(* Logix 5000 project; controller DIMTER vendor 1 type 14 code 77 rev 15.4; software revision 15.01 *)
// Dimter PLC Upgrade

TASK MainTask (continuous, watchdog 500 ms) : MainProgram

MODULES
   Controller : vendor 1 type 14 code 77 (CompactLogixL32EController 0, rev 15.4)
      LocalENB : 1769-L32E Ethernet Port (CompactLogixL32Ethernet 1, Ethernet 10.1.1.1, rev 15.1)
      Local : CompactBus (CompactVirtualAdapter 3, rev 15.1, Input RPI 2 ms)
          : 1769-IQ32 (Compact 1, rev 3.1, Input RPI 2 ms)
          : 1769-IQ32 (Compact 2, rev 3.1, Input RPI 2 ms)
          : 1769-IQ32 (Compact 3, rev 3.1, Input RPI 2 ms)
          : 1769-OW16 (Compact 4, rev 1.1, Output RPI 2 ms)
          : 1769-OW16 (Compact 5, rev 1.1, Output RPI 2 ms)
          : 1769-OW16 (Compact 6, rev 1.1, Output RPI 2 ms)
          : 1769-OW16 (Compact 7, rev 1.1, Output RPI 2 ms)
END_MODULES

TYPE FaultRecord :
STRUCT
   TimeLow : DINT;
   TimeHigh : DINT;
   Type : INT;
   Code : INT;
   Info : DINT[8];
END_STRUCT
END_TYPE

TYPE RTC :   // Real Time Clock
STRUCT
   Year : DINT;   // RTC Year
   Month : DINT;   // RTC Month
   Day : DINT;   // RTC Day
   Hour : DINT;   // RTC Hour
   Minute : DINT;   // RTC Minute
   Second : DINT;   // RTC Second
   uSecond : DINT;   // RTC uSecond
   DayOfWeek : DINT;   // RTC Day Of Week
END_STRUCT
END_TYPE

VAR_GLOBAL   (* controller tags *)
   A120 : ALIAS FOR Local:4:O.Data.0;   // O:4.0/0 A12.0 Buffer Selection1
   A121 : ALIAS FOR Local:4:O.Data.1;   // O:4.0/1 A12/1 Buffer Selection 2
   A122 : ALIAS FOR Local:4:O.Data.2;   // O:4.0/2 A12.2 Reset Failure
   A123 : ALIAS FOR Local:4:O.Data.3;   // O:4.0/3 A12.3 Reset Buffer
   A124 : ALIAS FOR Local:4:O.Data.4;   // O:4.0/4 A12.4 Spare
   A125 : ALIAS FOR Local:4:O.Data.5;   // O:4.0/5 A12.5 Spare
   A126 : ALIAS FOR Local:4:O.Data.6;   // O:4.0/6 A12.6 Spare
   A127 : ALIAS FOR Local:4:O.Data.7;   // O:4.0/7 A12.7 Spare
   A130 : ALIAS FOR Local:4:O.Data.8;   // O:4.0/8 A13.0 Failure Conveyor
   A131 : ALIAS FOR Local:4:O.Data.9;   // O:4.0/9 A13.1 Failure Saw 1
   A132 : ALIAS FOR Local:4:O.Data.10;   // O:4.0/10 A13.2 Failure Saw 2
   A133 : ALIAS FOR Local:4:O.Data.11;   // O:4.0/11 A13.3 Defect Measuring Computer
   A134 : ALIAS FOR Local:4:O.Data.12;   // O:4.0/12 A13.4 Safety Barrier Transfer Station
   A135 : ALIAS FOR Local:4:O.Data.13;   // O:4.0/13 A13.5 Unknown
   A136 : ALIAS FOR Local:4:O.Data.14;   // O:4.0/14 A136 Unknown
   A137 : ALIAS FOR Local:4:O.Data.15;   // O:4.0/15 A137 Safety Barrier Transfer Station
   A140 : ALIAS FOR Local:5:O.Data.0;   // O:5.0/0 A140 Chain Ejector Fast Left
   A141 : ALIAS FOR Local:5:O.Data.1;   // O:5.0/1 A141 Chain Ejector Slow Left
   A142 : ALIAS FOR Local:5:O.Data.2;   // O:5.0/2 A142 Raise Rake 1
   A143 : ALIAS FOR Local:5:O.Data.3;   // O:5.0/3 A143 Brake Cross Conveyor Front of Saw 1
   A144 : ALIAS FOR Local:5:O.Data.4;   // O:5.0/4 A144 Cross Feed 1 Fast Fwd
   A145 : ALIAS FOR Local:5:O.Data.5;   // O:5.0/5 A145 Cross Feed 1 Slow Fwd
   A146 : ALIAS FOR Local:5:O.Data.6;   // O:5.0/6 A146 Cross Feed 1 Fast Rev
   A147 : ALIAS FOR Local:5:O.Data.7;   // O:5.0/7 A147 Infeed Roller Saw 1
   A150 : ALIAS FOR Local:5:O.Data.8;   // O:5.0/8 A15.0 Rollcase 1 VSD Run Enable
   A151 : ALIAS FOR Local:5:O.Data.9;   // O:5.0/9 A15.1 Jog Rollcase 1 Set Speed
   A152 : ALIAS FOR Local:5:O.Data.10;   // O:5.0/10 A15.2 Forward Rotation Rollcase 1
   A153 : ALIAS FOR Local:5:O.Data.11;   // O:5.0/11 A15.3 Brake Rollcase Front of Saw 1
   A154 : ALIAS FOR Local:5:O.Data.12;   // O:5.0/12 A15.4 Rollcase 2 VSD Run Enable
   A155 : ALIAS FOR Local:5:O.Data.13;   // O:5.0/13 A155 Jog Rollcase 2 Set Speed
   A156 : ALIAS FOR Local:5:O.Data.14;   // O:5.0/14 A156 Forward Rotation Rollcase 2
   A157 : ALIAS FOR Local:5:O.Data.15;   // O:5.0/15 A157 Brake Rollcase 2
   A160 : ALIAS FOR Local:6:O.Data.0;   // O:6.0/0 A16.0 Chain Ejector Fast Right
   A161 : ALIAS FOR Local:6:O.Data.1;   // O:6.0/1 A16.1 Chain Ejector Slow Right
   A162 : ALIAS FOR Local:6:O.Data.2;   // O:6.0/2 A16.2 Rake 2
   A163 : ALIAS FOR Local:6:O.Data.3;   // O:6.0/3 A16.3 Brake Cross Conveyor Front of Saw 2
   A164 : ALIAS FOR Local:6:O.Data.4;   // O:6.0/4 A16.4 Cross Feed 2 Fast Fwd
   A165 : ALIAS FOR Local:6:O.Data.5;   // O:6.0/5 A16.5 Cross Feed 2 Slow Fwd
   A166 : ALIAS FOR Local:6:O.Data.6;   // O:6.0/6 A16.6 Cross Feed 2 Fast Rev
   A167 : ALIAS FOR Local:6:O.Data.7;   // O:6.0/7 A16.7 Infeed Roller Saw 2
   A170 : ALIAS FOR Local:6:O.Data.8;   // O:6.0/8 A17.0 Infeed Measuring Slot Weinig Release Workpiece to Demand
   A171 : ALIAS FOR Local:6:O.Data.9;   // O:6.0/9 A17.1 Conveyor Measuring Slot Weinig Feed to Switch On
   A172 : ALIAS FOR Local:6:O.Data.10;   // O:6.0/10 A17.2 Chain Ejector Brake
   A173 : ALIAS FOR Local:6:O.Data.11;   // O:6.0/11 A17.3 Spare
   A174 : ALIAS FOR Local:6:O.Data.12;   // O:6.0/12 A17.4 Spare
   A175 : ALIAS FOR Local:6:O.Data.13;   // O:6.0/13 A17.5 Spare
   A176 : ALIAS FOR Local:6:O.Data.14;   // O:6.0/14 A17.6 Spare
   A177 : ALIAS FOR Local:6:O.Data.15;   // O:6.0/15 A17.7 Spare
   A180 : ALIAS FOR Local:7:O.Data.0;   // O:7.0/0 A18.0 VSD Feed Contactor Rollcase 1
   A181 : ALIAS FOR Local:7:O.Data.1;   // O:7.0/1 A18.1 VSD Feed Contactor Rollcase 2
   A182 : ALIAS FOR Local:7:O.Data.2;   // O:7.0/2 A18.2 Infeed Roller Measuring Station
   A183 : ALIAS FOR Local:7:O.Data.3;   // O:7.0/3 A18.3 Unknown
   A184 : ALIAS FOR Local:7:O.Data.4;   // O:7.0/4 A18.4 Waste Belt Conveyor 1
   A185 : ALIAS FOR Local:7:O.Data.5;   // O:7.0/5 A18.5 Waste Belt Conveyor 2
   A186 : ALIAS FOR Local:7:O.Data.6;   // O:7.0/6 A18.6 Cross Belt 1
   A187 : ALIAS FOR Local:7:O.Data.7;   // O:7.0/7 A18.7 Cross Belt 2
   A190 : ALIAS FOR Local:7:O.Data.8;   // O:7.0/8 A19.0 Spare
   A191 : ALIAS FOR Local:7:O.Data.9;   // O:7.0/9 A19.1 Spare
   A192 : ALIAS FOR Local:7:O.Data.10;   // O:7.0/10 A19.2 Spare
   A193 : ALIAS FOR Local:7:O.Data.11;   // O:7.0/11 A19.3 Spare
   A194 : ALIAS FOR Local:7:O.Data.12;   // O:7.0/12 A19.4 Spare
   A195 : ALIAS FOR Local:7:O.Data.13;   // O:7.0/13 A19.5 Spare
   A196 : ALIAS FOR Local:7:O.Data.14;   // O:7.0/14 A19.6 Spare
   A197 : ALIAS FOR Local:7:O.Data.15;   // O:7.0/15 A19.7 Spare
   BitArrayFromHMI : INT[100]; {produced}
   BitArrayToHMI : INT[130] := ([6] := 14, [7] := 15);
   BitsFromHMI : BOOL[128];   // Bits From HMI
   Debounce : TIMER[30] := ([0].PRE := 100, [1].PRE := 100);   // Debounce Timers
        [0]   // PE Infeed Saw 1 Debounce
        [1]   // PE Roller 1 Debounce
   Delay : TIMER[30] := ([0].PRE := 300, [1].PRE := 300, [2].PRE := 100);   // Delay Timers
        [0]   // Saw 1 Cutting Delay
        [1]   // Saw 2 Cutting Delay
   E00 : ALIAS FOR Local:1:I.Data.0;   // I:1.0/0 E0.0 Control Power On
   E01 : ALIAS FOR Local:1:I.Data.1;   // I:1.0/1 E0.1 Saw Hood 1 Closed
   E02 : ALIAS FOR Local:1:I.Data.2;   // I:1.0/2 E0.2 Saw Motor 1 On
   E03 : ALIAS FOR Local:1:I.Data.3;   // I:1.0/3 E0.3 Release - Feed Saw 1
   E04 : ALIAS FOR Local:1:I.Data.4;   // I:1.0/4 E0.4 Failure Saw 1
   E05 : ALIAS FOR Local:1:I.Data.5;   // I:1.0/5 E0.5 Failure Chain Ejector
   E06 : ALIAS FOR Local:1:I.Data.6;   // I:1.0/6 E0.6 Failure Conveyor in Front of Saw 1
   E07 : ALIAS FOR Local:1:I.Data.7;   // I:1.0/7 E0.7 Failure Conveyor in Front of Saw 2
   E10 : ALIAS FOR Local:1:I.Data.8;   // I:1.0/8 E1.0 Failure Weinig Conveyor
   E100 : ALIAS FOR Local:3:I.Data.16;   // I:3.1/0 E10.0 Sorting Ejector Sorting 1
   E101 : ALIAS FOR Local:3:I.Data.17;   // I:3.1/1 E10.1 Sorting Ejector 2 Sorting 1
   E102 : ALIAS FOR Local:3:I.Data.18;   // I:3.1/2 E10.2 Sorting Ejector 3 Sorting 1
   E103 : ALIAS FOR Local:3:I.Data.19;   // I:3.1/3 E10.3 Sorting Ejector 1 Sorting 2
   E104 : ALIAS FOR Local:3:I.Data.20;   // I:3.1/4 E10.4 Sorting Ejector 2 Sorting 2
   E105 : ALIAS FOR Local:3:I.Data.21;   // I:3.1/5 E10.5 Sorting Ejector 3 Sorting 2
   E106 : ALIAS FOR Local:3:I.Data.22;   // I:3.1/6 E10.6 Cross Belt 1 Cyclewise Continuous Running
   E107 : ALIAS FOR Local:3:I.Data.23;   // I:3.1/7 E10.7 ???
   E11 : ALIAS FOR Local:1:I.Data.9;   // I:1.0/9 E1.1 Saw Hood 2 Closed
   E110 : ALIAS FOR Local:3:I.Data.24;   // I:3.1/8 E11.0 Cross Belt 1 Footswitch (Removed)
   E111 : ALIAS FOR Local:3:I.Data.25;   // I:3.1/9 E11.1 Cross Belt 2 Cyclewise Continuous Running
   E112 : ALIAS FOR Local:3:I.Data.26;   // I:3.1/10 E11.2 ???
   E113 : ALIAS FOR Local:3:I.Data.27;   // I:3.1/11 E11.3 Cross Belt 2 Footswitch (Removed)
   E114 : ALIAS FOR Local:3:I.Data.28;   // I:3.1/12 E11.4 Transfer Station On
   E115 : ALIAS FOR Local:3:I.Data.29;   // I:3.1/13 E11.5 Cross Feed Manual Fwd-Rev
   E116 : ALIAS FOR Local:3:I.Data.30;   // I:3.1/14 E11.6 ???
   E117 : ALIAS FOR Local:3:I.Data.31;   // I:3.1/1 5 E11.7 Acknowledge Failure
   E12 : ALIAS FOR Local:1:I.Data.10;   // I:1.0/10 E1.2 Saw Motor 2 On
   E13 : ALIAS FOR Local:1:I.Data.11;   // I:1.0/11 E1.3 Release - Feed Saw 2
   E14 : ALIAS FOR Local:1:I.Data.12;   // I:1.0/12 E1.4 Failure Saw 2
   E15 : ALIAS FOR Local:1:I.Data.13;   // I:1.0/13 E1.5 Data Ready At Saw
   E16 : ALIAS FOR Local:1:I.Data.14;   // I:1.0/14 E1.6 Release Optimisation
   E17 : ALIAS FOR Local:1:I.Data.15;   // I:1.0/15 E1.7 Defect Measuring Computer
   E20 : ALIAS FOR Local:1:I.Data.16;   // I:1.1/0 E2.0 Protection Hood Measuring System
   E21 : ALIAS FOR Local:1:I.Data.17;   // I:1.1/1 E2.1 Spare
   E22 : ALIAS FOR Local:1:I.Data.18;   // I:1.1/2 E2.2 Frequency Converter Rollcase in Front of Saw 1 Ready For Operation
   E23 : ALIAS FOR Local:1:I.Data.19;   // I:1.1/3 E2.3 Frequency Converter Rollcase in Front of Saw 2 Ready For Operation
   E24 : ALIAS FOR Local:1:I.Data.20;   // I:1.1/4 E2.4 Emergency Shutdown Internal
   E25 : ALIAS FOR Local:1:I.Data.21;   // I:1.1/5 E2.5 Emergency Shutdown External
   E26 : ALIAS FOR Local:1:I.Data.22;   // I:1.1/6 E2.6 Safety Barrier at Transfer Station Closed
   E27 : ALIAS FOR Local:1:I.Data.23;   // I:1.1/7 E2.7 Reset Safety Barrier at Transfer Station
   E30 : ALIAS FOR Local:1:I.Data.24;   // I:1.1/8 E3.0 Spare
   E31 : ALIAS FOR Local:1:I.Data.25;   // I:1.1/9 E3.1 PE in Front of Measuring Station
   E32 : ALIAS FOR Local:1:I.Data.26;   // I:1.1/10 E3.2 Start Measurement Measurement Station
   E33 : ALIAS FOR Local:1:I.Data.27;   // I:1/1/11 E3.3 PE Behind Measurement Station
   E34 : ALIAS FOR Local:1:I.Data.28;   // I:1.1/12 E3.4 Spare
   E35 : ALIAS FOR Local:1:I.Data.29;   // I:1.1/13 E3.5 Spare
   E36 : ALIAS FOR Local:1:I.Data.30;   // I:1.1/14 E3.6 Spare
   E37 : ALIAS FOR Local:1:I.Data.31;   // I:1.1/15 E3.7 Spare
   E40 : ALIAS FOR Local:2:I.Data.0;   // I:2.0/0 E4.0 Chain Ejector Manual Left
   E41 : ALIAS FOR Local:2:I.Data.1;   // I:2.0/1 E4.1 Cross Feed 1 Manual Fwd - Rev
   E42 : ALIAS FOR Local:2:I.Data.2;   // I:2.0/2 E4.2 Cross Feed 1 Manual Fwd - Rev
   E43 : ALIAS FOR Local:2:I.Data.3;   // I:2.0/3 E4.3 Infeed Saw 1 On
   E44 : ALIAS FOR Local:2:I.Data.4;   // I:2.0/4 E4.4 Waste Conveyor Belt On
   E45 : ALIAS FOR Local:2:I.Data.5;   // I:2.0/5 E4.5 Transfer Station in Front of Saw On
   E46 : ALIAS FOR Local:2:I.Data.6;   // I:2.0/6 E4.6 Acknowledge Failure
   E47 : ALIAS FOR Local:2:I.Data.7;   // I:2.0/7 E4.7 Lamp Test
   E50 : ALIAS FOR Local:2:I.Data.8;   // I:2.0/8 E5.0 Chain Ejector Manual Right
   E51 : ALIAS FOR Local:2:I.Data.9;   // I:2.0/9 E5.1 Cross Feed 2 Manual Fwd - Rev
   E52 : ALIAS FOR Local:2:I.Data.10;   // I:2.0/10 E5.2 Cross Feed 2 Manual Fwd - Rev
   E53 : ALIAS FOR Local:2:I.Data.11;   // I:2.0/11 E5.3 Infeed Saw 2 On
   E54 : ALIAS FOR Local:2:I.Data.12;   // I:2.0/12 E5.4 Measuring Station On
   E55 : ALIAS FOR Local:2:I.Data.13;   // I:2.0/13 E5.5 Reset Defect Measuring Computer
   E56 : ALIAS FOR Local:2:I.Data.14;   // I:2.0/14 E5.6 Reset Buffer Measuring Computer
   E57 : ALIAS FOR Local:2:I.Data.15;   // I:2.0/15 E5.7 Conveyor Measuring Station Manual
   E60 : ALIAS FOR Local:2:I.Data.16;   // I:2.1/0 E6.0 Spare
   E61 : ALIAS FOR Local:2:I.Data.17;   // I:2.1/1 E6.1 PE Infeed Saw 1
   E62 : ALIAS FOR Local:2:I.Data.18;   // I:2.1/2 E6.2 PE Front of Saw 1
   E63 : ALIAS FOR Local:2:I.Data.19;   // I:2.1/3 E6.3 PE Roller 1
   E64 : ALIAS FOR Local:2:I.Data.20;   // I:2.1/4 E6.4 Feed Saw 1 On
   E65 : ALIAS FOR Local:2:I.Data.21;   // I:2.1/5 E6.5 Spare
   E66 : ALIAS FOR Local:2:I.Data.22;   // I:2.1/6 E6.6 Release Chain Ejector Saw 1 Cross Feed
   E67 : ALIAS FOR Local:2:I.Data.23;   // I:2.1/7 E6.7 PE Cross Feed 1 Waiting Position
   E70 : ALIAS FOR Local:2:I.Data.24;   // I:2.1/8 E7.0 PE Chain Ejector Home Position Left
   E71 : ALIAS FOR Local:2:I.Data.25;   // I:2.1/9 E7.1 PE Chain Ejector Initial Position Left Front
   E72 : ALIAS FOR Local:2:I.Data.26;   // I:2.1/10 E7.2 Stop Rollcase 1
   E73 : ALIAS FOR Local:2:I.Data.27;   // I:2.1/11 E7.3 Cross Feed 1 Down
   E74 : ALIAS FOR Local:2:I.Data.28;   // I:2.1/12 E7.4 Cross Feed 1 Up
   E75 : ALIAS FOR Local:2:I.Data.29;   // I:2.1/13 E7.5 Cross Feed 1 Initial Position
   E76 : ALIAS FOR Local:2:I.Data.30;   // I:2.1/14 E7.6 PE Cross Feed 1 Slow Fwd
   E77 : ALIAS FOR Local:2:I.Data.31;   // I:2.1/15 E7.7 Cross Feed 1 at Front
   E80 : ALIAS FOR Local:3:I.Data.0;   // I:3.0/0 E8.0 Spare
   E81 : ALIAS FOR Local:3:I.Data.1;   // I:3.0/1 E8.1 PE Infeed Saw 2
   E82 : ALIAS FOR Local:3:I.Data.2;   // I:3.0/2 E8.2 PE Front of Saw 2
   E83 : ALIAS FOR Local:3:I.Data.3;   // I:3.0/3 E8.3 PE Roller 2
   E84 : ALIAS FOR Local:3:I.Data.4;   // I:3.0/4 E8.4 Feed Saw 2 On
   E85 : ALIAS FOR Local:3:I.Data.5;   // I:3.0/5 E8.5 Spare
   E86 : ALIAS FOR Local:3:I.Data.6;   // I:3.0/6 E8.6 Release (Enable) Chain Ejector Saw 2 Cross Feed
   E87 : ALIAS FOR Local:3:I.Data.7;   // I:3.0/7 E8.7 PE Cross Feed 2 Waiting Position
   E90 : ALIAS FOR Local:3:I.Data.8;   // I:3.0/8 E9.0 PE Chain Ejector Initial Position Right
   E91 : ALIAS FOR Local:3:I.Data.9;   // I:3.0/9 E9.1 PE Chain Ejector Initial Position Right Front
   E92 : ALIAS FOR Local:3:I.Data.10;   // I:3.0/10 E9.2 Stop Rollcase 2
   E93 : ALIAS FOR Local:3:I.Data.11;   // I:3.0/11 E9.3 Cross Feed 2 Down
   E94 : ALIAS FOR Local:3:I.Data.12;   // I:3.0/12 E9.4 Cross Feed 2 Up
   E95 : ALIAS FOR Local:3:I.Data.13;   // I:3.0/13 E9.5 Cross Feed 2 Home Position
   E96 : ALIAS FOR Local:3:I.Data.14;   // I:3.0/14 E9.6 PE Cross Feed 2 Slow Fwd
   E97 : ALIAS FOR Local:3:I.Data.15;   // I:3.0/15 E9.7 Cross Feed 2 at Front
   Faults : BOOL[224] := ([0] := 1, [14] := 1);   // Fault Array
   FirstPass : BOOL;   // On for First Scan
   HMI_Bits : BOOL[2016] := ([20] := 1, [44] := 1, [111] := 1, [112] := 1, [113] := 1, [114] := 1, [115] := 1, [118] := 1, [119] := 1, [120] := 1, [121] := 1, [122] := 1, [316] := 1, [330] := 1, [357] := 1, [1033] := 1); {produced}   // Bits to HMI
   HMI_IntWords : INT[200] := ([0] := 38, [2] := 323, [3] := 268, [4] := 591, [30] := 427, [31] := 576, [32] := 1003, [34] := 403, [35] := 649, [36] := 1052, [38] := 1543, [39] := 1599, [40] := 3142, [42] := 374, [43] := 450, [44] := 824, [46] := 1739, [47] := 1704, [48] := 3443, [54] := 2187, [55] := 2818, [56] := 5005, [58] := 427, [59] := 576, [60] := 1003, [62] := 403, [63] := 649, [64] := 1052, [66] := 1543, [67] := 1599, [68] := 3142, [70] := 374, [71] := 450, [72] := 824, [74] := 1739, [75] := 1704, [76] := 3443, [82] := 2187, [83] := 2818, [84] := 5005); {produced}   // Integer Words to HMI
        [0]   // Screen Command to HMI
        [1]   // Screen Displayed From HMI
        [2]   // Shift A Monday Saw 1 Total
        [3]   // Shift A Monday Saw 2 Total
        [4]   // Shift A Monday Grand Total
        [5]   // Shift A Monday Total Faults
        [6]   // Shift A Tuesday Saw 1 Total
        [7]   // Shift A Tuesday Saw 2 Total
        [8]   // Shift A Tuesday Grand Total
        [9]   // Shift A Tuesday Total Faults
        [10]   // Shift A Wednesday Saw 1 Total
        [11]   // Shift A Wednesday Saw 2 Total
        [12]   // Shift A Wednesday Grand Total
        [13]   // Shift A Wednesday Total Faults
        [14]   // Shift A Thursday Saw 1 Total
        [15]   // Shift A Thursday Saw 2 Total
        [16]   // Shift A Thursday Grand Total
        [17]   // Shift A Thursday Total Faults
        [18]   // Shift A Friday Saw 1 Total
        [19]   // Shift A Friday Saw 2 Total
        [20]   // Shift A Friday Grand Total
        [21]   // Shift A Friday Total Faults
        [22]   // Shift A Saturday Saw 1 Total
        [23]   // Shift A Saturday Saw 2 Total
        [24]   // Shift A Saturday Grand Total
        [25]   // Shift A Saturday Total Faults
        [26]   // Shift A Sunday Saw 1 Total
        [27]   // Shift A Sunday Saw 2 Total
        [28]   // Shift A Sunday Grand Total
        [29]   // Shift A Sunday Total Faults
        [30]   // Shift B Monday Saw 1 Total
        [31]   // Shift B Monday Saw 2 Total
        [32]   // Shift B Monday Grand Total
        [33]   // Shift B Monday Total Faults
        [34]   // Shift B Tuesday Saw 1 Total
        [35]   // Shift B Tuesday Saw 2 Total
        [36]   // Shift B Tuesday Grand Total
        [37]   // Shift B Tuesday Total Faults
        [38]   // Shift B Wednesday Saw 1 Total
        [46]   // Shift B Friday Saw 1 Total
        [47]   // Shift B Friday Saw 2 Total
        [43]   // Shift B Thursday Saw 2 Total
        [48]   // Shift B Friday Grand Total
        [39]   // Shift B Wednesday Saw 2 Total
        [40]   // Shift B Wednesday Grand Total
        [41]   // Shift B Wednesday Total Faults
        [42]   // Shift B Thursday Saw 1 Total
        [44]   // Shift B Thursday Grand Total
        [45]   // Shift B Thursday Total Faults
        [49]   // Shift B Friday Total Faults
        [50]   // Shift B Saturday Saw 1 Total
        [51]   // Shift B Saturday Saw 2 Total
        [52]   // Shift B Saturday Grand Total
        [53]   // Shift B Saturday Total Faults
        [54]   // Shift B Sunday Saw 1 Total
        [55]   // Shift B Sunday Saw 2 Total
        [56]   // Shift B Sunday Grand Total
        [57]   // Shift B Sunday Total Faults
        [58]   // Shift C Monday Saw 1 Total
        [59]   // Shift C Monday Saw 2 Total
        [60]   // Shift C Monday Grand Total
        [61]   // Shift C Monday Total Faults
        [62]   // Shift C Tuesday Saw 1 Total
        [63]   // Shift C Tuesday Saw 2 Total
        [64]   // Shift C Tuesday Grand Total
        [65]   // Shift C Tuesday Total Faults
        [66]   // Shift C Wednesday Saw 1 Total
        [67]   // Shift C Wednesday Saw 2 Total
        [68]   // Shift C Wednesday Grand Total
        [69]   // Shift C Wednesday Total Faults
        [70]   // Shift C Thursday Saw 1 Total
        [71]   // Shift C Thursday Saw 2 Total
        [72]   // Shift C Thursday Grand Total
        [73]   // Shift C Thursday Total Faults
        [74]   // Shift C Friday Saw 1 Total
        [75]   // Shift C Friday Saw 2 Total
        [76]   // Shift C Friday Grand Total
        [77]   // Shift C Friday Total Faults
        [78]   // Shift C Saturday Saw 1 Total
        [79]   // Shift C Saturday Saw 2 Total
        [80]   // Shift C Saturday Grand Total
        [81]   // Shift C Saturday Total Faults
        [82]   // Shift C Sunday Saw 1 Total
        [83]   // Shift C Sunday Saw 2 Total
        [84]   // Shift C Sunday Grand Total
        [85]   // Shift C Sunday Total Faults
   HMI_RealWords : REAL[20]; {produced}   // Real Words to HMI Transfer file
        [1]   // Saw 2 Hourmeter
        [4]   // Cross Feed 1 Hourmeter
        [7]   // Waste Belt 1 Hourmeter
        [2]   // Infeed Rolls 1 Hourmeter
        [0]   // Saw 1 Hourmeter
        [3]   // Infeed Rolls 2 Hourmeter
        [5]   // Cross Feed 2 Hourmeter
        [6]   // Chain Ejector Hourmeter
        [8]   // Waste Belt 2 Hourmeter
        [9]   // Cross Belt 1 Hourmeter
        [10]   // Cross Belt 2 Hourmeter
   HMI_TimerPresets : INT[100]; {produced}   // Timer Preset Data from HMI
   IntsFromHMI : INT[100] := ([0] := 5, [2] := 13, [4] := 5, [6] := 13, [8] := 5, [10] := 13, [12] := 5, [14] := 13, [16] := 5, [18] := 13, [28] := 13, [30] := 23, [32] := 13, [34] := 23, [36] := 13, [38] := 23, [40] := 13, [42] := 23, [44] := 13, [46] := 23, [56] := 21, [58] := 5, [60] := 21, [62] := 5, [63] := 21, [65] := 5, [66] := 21, [68] := 5, [69] := 21, [71] := 5, [72] := 21, [74] := 5);   // Integers From HMI
        [0]   // Shift A Monday Start Hour
        [2]   // Shift A Monday Finish Hour
        [1]   // Shift A Monday Start Minute
        [3]   // Shift A Monday Finish Minute
        [4]   // Shift A Tuesday Start Hour
        [6]   // Shift A Tuesday Finish Hour
        [8]   // Shift A Wednesday Start Hour
        [5]   // Shift A Tuesday Start Minute
        [7]   // Shift A Tuesday Finish Minute
        [9]   // Shift A Wednesday Start Minute
        [10]   // Shift A Wednesday Finish Hour
        [11]   // Shift A Wednesday Finish Minute
        [12]   // Shift A Thursday Start Hour
        [13]   // Shift A Thursday Start Minute
        [14]   // Shift A Thursday Finish Hour
        [15]   // Shift A Thursday Finish Minute
        [16]   // Shift A Friday Start Hour
        [17]   // Shift A Friday Start Minute
        [18]   // Shift A Friday Finish Hour
        [19]   // Shift A Friday Finish Minute
        [20]   // Shift A Saturday Start Hour
        [21]   // Shift A Saturday Start Minute
        [22]   // Shift A Saturday Finish Hour
        [23]   // Shift A Saturday Finish Minute
        [24]   // Shift A Sunday Start Hour
        [25]   // Shift A Sunday Start Minute
        [26]   // Shift A Sunday Finish Hour
        [27]   // Shift A Sunday Finish Minute
        [28]   // Shift B Monday Start Hour
        [29]   // Shift B Monday Start Minute
        [30]   // Shift B Monday Finish Hour
        [31]   // Shift B Monday Finish Minute
        [32]   // Shift B Tuesday Start Hour
        [33]   // Shift B Tuesday Start Minute
        [34]   // Shift B Tuesday Finish Hour
        [35]   // Shift B Tuesday Finish Minute
        [36]   // Shift B Wednesday Start Hour
        [37]   // Shift B Wednesday Start Minute
        [38]   // Shift B Wednesday Finish Hour
        [39]   // Shift B Wednesday Finish Minute
        [40]   // Shift B Thursday Start Hour
        [41]   // Shift B Thursday Start Minute
        [42]   // Shift B Thursday Finish Hour
        [43]   // Shift B Thursday Finish Minute
        [44]   // Shift B Friday Start Hour
        [45]   // Shift B Friday Start Minute
        [46]   // Shift B Friday Finish Hour
        [47]   // Shift B Friday Finish Minute
        [48]   // Shift B Saturday Start Hour
        [49]   // Shift B Saturday Start Minute
        [50]   // Shift B Saturday Finish Hour
        [51]   // Shift B Saturday Finish Minute
        [52]   // Shift B Sunday Start Hour
        [53]   // Shift B Sunday Start Minute
        [54]   // Shift B Sunday Finish Hour
        [55]   // Shift B Sunday Finish Minute
        [56]   // Shift C Monday Start Hour
        [57]   // Shift C Monday Start Minute
        [58]   // Shift C Monday Finish Hour
        [59]   // Shift C Monday Finish Minute
        [60]   // Shift C Tuesday Start Hour
        [61]   // Shift C Tuesday Start Minute
        [62]   // Shift C Tuesday Finish Hour
        [63]   // Shift C Tuesday Finish Minute
        [64]   // Shift C Wednesday Start Hour
        [65]   // Shift C Wednesday Start Minute
        [66]   // Shift C Wednesday Finish Hour
        [67]   // Shift C Wednesday Finish Minute
        [68]   // Shift C Thursday Start Hour
        [69]   // Shift C Thursday Start Minute
        [70]   // Shift C Thursday Finish Hour
        [71]   // Shift C Thursday Finish Minute
        [72]   // Shift C Friday Start Hour
        [73]   // Shift C Friday Start Minute
        [74]   // Shift C Friday Finish Hour
        [75]   // Shift C Friday Finish Minute
        [76]   // Shift C Saturday Start Hour
        [77]   // Shift C Saturday Start Minute
        [78]   // Shift C Saturday Finish Hour
        [82]   // Shift C Sunday Finish Hour
        [80]   // Shift C Sunday Start Hour
        [79]   // Shift C Saturday Finish Minute
        [81]   // Shift C Sunday Start Minute
        [83]   // Shift C Sunday Finish Minute
   RealTimeClock : DINT[10] := ([0] := 2006, [1] := 7, [2] := 21, [3] := 16, [4] := 13, [5] := 8, [6] := 204124, [7] := 5);
        [0]   // RTC Year
        [1]   // RTC Month
        [2]   // RTC Day
        [3]   // RTC Hour
        [4]   // RTC Minute
        [5]   // RTC Second
        [6]   // RTC uSecond
        [7]   // RTC Day Of Week
   Status : BOOL[224] := ([0] := 1);   // Status Array
END_VAR

PROGRAM FaultHandler   (* main routine Main *)
VAR
   LastMajorFaultRecord : DINT;
   Major_Fault_Record : FaultRecord;
END_VAR

ROUTINE Main   (* ladder *)
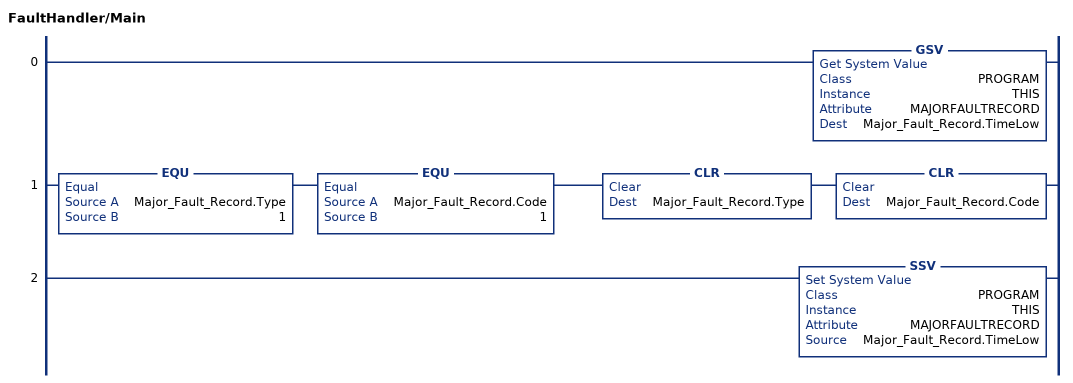
   0: GSV(PROGRAM,THIS,MAJORFAULTRECORD,Major_Fault_Record.TimeLow);
   1: EQU(Major_Fault_Record.Type,1)EQU(Major_Fault_Record.Code,1)CLR(Major_Fault_Record.Type)CLR(Major_Fault_Record.Code);
   2: SSV(PROGRAM,THIS,MAJORFAULTRECORD,Major_Fault_Record.TimeLow);
END_ROUTINE
END_PROGRAM

PROGRAM FirstPass   (* main routine FirstPass *)
VAR
   Major_Fault_Record : FaultRecord := (TimeLow := -190438328, TimeHigh := 253875, Info[0] := -1873559692, Info[1] := 253870);
END_VAR

ROUTINE FirstPass   (* ladder *)
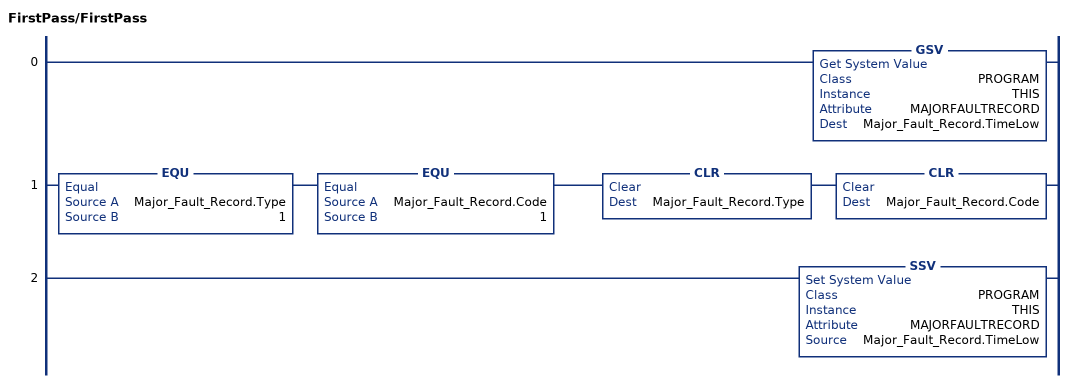
   0: GSV(PROGRAM,THIS,MAJORFAULTRECORD,Major_Fault_Record.TimeLow);
   1: EQU(Major_Fault_Record.Type,1)EQU(Major_Fault_Record.Code,1)CLR(Major_Fault_Record.Type)CLR(Major_Fault_Record.Code);
   2: SSV(PROGRAM,THIS,MAJORFAULTRECORD,Major_Fault_Record.TimeLow);
END_ROUTINE
END_PROGRAM

PROGRAM MainProgram   (* main routine MainRoutine *)
VAR
   Bit_FIFO_Control : CONTROL;
   BufferReady : TIMER := (PRE := 15000);
   ChainEjectorRunHourTimer : TIMER := (PRE := 360000);   // Chain Ejector Run Hourmeter 1/10th Hour Timer
   CrossBelt1RunHourTimer : TIMER := (PRE := 360000);   // Cross Belt 1 Run Hourmeter 1/10th Hour Timer
   CrossBelt2RunHourTimer : TIMER := (PRE := 360000);   // Cross Belt 2 Run Hourmeter 1/10th Hour Timer
   CrossFeed1RunHourTimer : TIMER := (PRE := 360000);   // Cross Feed 1 Run Hourmeter 1/10th Hour Timer
   CrossFeed2RunHourTimer : TIMER := (PRE := 360000);   // Cross Feed 2 Run Hourmeter 1/10th Hour Timer
   CurrentShift : DINT := 2;   // Shift Currently Operating
   DisplaySplashScreen : BOOL;
   F : BOOL[2016] := ([44] := 1, [111] := 1, [112] := 1, [113] := 1, [114] := 1, [115] := 1, [118] := 1, [119] := 1, [120] := 1, [121] := 1, [122] := 1, [316] := 1, [1033] := 1);   // Flags
        [997]   // Both Saws Are Running
        [370]   // Timber In Saw 1
        [307]   // Buffering to Saw 2
        [1370]   // Timber In Saw 2
        [291]   // Measuring Computer In Use
        [302]   // Only Saw 2 Available For Selection
        [380]   // Saw 1 Servo Drive Feeding
        [326]   // Chain Ejector Watchdog fault
        [360]   // Reset Saw 1 Timber At Infeed
        [444]   // Cross Belt 1 Run
        [1322]   // Chain Ejector Run Fast Right
        [322]   // Chain Ejector Run Fast Left
        [330]   // Transfer Stations On
        [20]   // Measuring Station On
        [45]   // Measuring Computer Begin Measuring
        [1023]   // Saw 1 Infeed Running
        [1327]   // Cross Feed 2 In Motion
        [310]   // Signal Saw Computer to Buffer Data to Saw 2
        [363]   // Saw 1 Timber At Saw
        [1362]   // Saw 2 Timber At Infeed
        [2009]   // Transfer Station Not On
        [450]   // Sorting Ejector 1 or 2 In Use
        [2011]   // Measuring Station Not On
        [292]   // Chain Ejector Running Fast
        [474]   // Cross Belt 2 Run
        [323]   // Chain Ejector Left Cycle Slow Down To Stop
        [1320]   // PLC Pulse to Saw Computer for Buffer to Saw 2 Complete
        [1336]   // Rollcase 2 Stopping (2)
        [313]   // Select Saw 2 For Buffer
        [40]   // Measuring Computer Failure
        [304]   // Buffering to Saw 1
        [1335]   // Timber on Cross Feed 2 Stop Sensor Stop Rollcase 2
        [321]   // Chain Ejector Run Left Manual
        [336]   // Rollcase 1 Stopping (2)
        [327]   // Cross Feed 1 In Motion
        [335]   // Timber on Cross Feed 1 Stop Sensor Stop Rollcase 1
        [1323]   // Chain Ejector Right Cycle Slow Down To Stop
        [340]   // Rollcase 1 Stopping (3)
        [1331]   // Chain Ejector Right Cycle Moving Slow
        [331]   // Chain Ejector Left Cycle Moving Slow
        [316]   // Chain Ejector Ejecting to Saw 2
        [305]   // Signal Saw Computer to Buffer Data to Saw 1
        [1321]   // Chain Ejector Run Right Manual
        [480]   // Sorting Ejector 3 In Use
        [1360]   // Reset Saw 2 Timber At Infeed
        [1380]   // Saw 2 Servo Drive Feeding
        [2012]   // Saw 2 Infeed Not Running
        [1363]   // Saw 2 Timber At Saw
        [50]   // Measurement Timing Complete
        [357]   // Safety Barrier Transfer Station OK
        [297]   // Measurement Complete
        [300]   // Both Saws Available For Selection
        [311]   // Select Saw 1 For Buffer
        [44]   // Measuring Computer OK
        [46]   // Begin Timing Measurement
        [301]   // Only Saw 1 Available For Selection
        [315]   // Chain Ejector Ejecting to Saw 1
        [362]   // Saw 1 Timber At Infeed
        [303]   // Buffer to Saw 1 Chain Ejector to Eject Left
        [306]   // Buffer to Saw 2 Chain Ejector to Eject Right
        [320]   // PLC Pulse to Saw Computer for Buffer to Saw 1 Complete
        [441]   // Cross Belt 1 Manual Run
        [470]   // Cross Belt 2 Manual Run
        [471]   // Cross Belt 2 Running Pulse
        [100]   // Saw 1 Hourmeter Reset Bit From HMI
        [101]   // Saw 2 Hourmeter Reset Bit From HMI
        [102]   // Infeed Rollcase 1 Hourmeter Reset Bit From HMI
        [103]   // Infeed Rollcase 2 Hourmeter Reset Bit From HMI
        [104]   // Cross Feed 1 Hourmeter Reset Bit From HMI
        [105]   // Cross Feed 2 Hourmeter Reset Bit From HMI
        [106]   // Chain Ejector Hourmeter Reset Bit From HMI
        [107]   // Waste Belt 1 Hourmeter Reset Bit From HMI
        [108]   // Waste Belt 2 Hourmeter Reset Bit From HMI
        [109]   // Cross Belt 1 Hourmeter Reset Bit From HMI
        [110]   // Cross Belt 2 Hourmeter Reset Bit From HMI
        [111]   // Shift A Monday Enable
        [112]   // Shift A Tuesday Enable
        [124]   // Shift B Sunday Enable
        [114]   // Shift A Thursday Enable
        [116]   // Shift A Saturday Enable
        [118]   // Shift B Monday Enable
        [117]   // Shift A Sunday Enable
        [115]   // Shift A Friday Enable
        [113]   // Shift A Wednesday Enable
        [119]   // Shift B Tuesday Enable
        [120]   // Shift B Wednesday Enable
        [121]   // Shift B Thursday Enable
        [122]   // Shift B Friday Enable
        [123]   // Shift B Saturday Enable
        [125]   // Shift C Monday Enable
        [126]   // Shift C Tuesday Enable
        [127]   // Shift C Wednesday Enable
        [128]   // Shift C Thursday Enable
        [129]   // Shift C Friday Enable
        [130]   // Shift C Saturday Enable
        [131]   // Shift C Sunday Enable
        [2000]   // Measuring Station Outfeed Blocked
        [2008]   // Saw 2 Infeed Blocked
        [1341]   // Rollcase 2 Has Stopped Cross Feed 2 Rake is Raised
        [341]   // Rollcase 1 Has Stopped Cross Feed 1 Rake Raised
        [1123]   // Saw 2 Infeed Running
        [1340]   // Rollcase 2 Stopping (3)
        [1345]   // Cross Feed 2 Running Manual
        [1344]   // Timber Ready at Saw 2
        [364]   // Cross Feed 1 Watchdog Timer Timed Out
        [1364]   // Cross Feed 2 Watch Dog Timer Fault
        [1033]   // Infeed for Saw 2 is On
        [345]   // Cross Feed 1 Running Manual
        [344]   // Timber Ready at Saw 1
        [1334]   // Raise Rake 2
        [334]   // Raise Rake 1
        [346]   // Saw 1 Timber Ready
        [1346]   // Saw 2 Timber Ready
   F312 : BOOL;   // Saw 1 Selected For Buffer
   F314 : BOOL;   // Saw 2 Selected For Buffer
   FlagTransferIndex : DINT := 126;   // Index Register For Copying Flags to HMI Files
   FlagTransferIndex2 : DINT := 6;
   FlagTransferIndex3 : DINT := 185;
   FlagTransferIndex4 : DINT;
   FLASHER : TIMER := (PRE := 500, ACC := 502, EN := 1, DN := 1);   // Lamp Flasher
   FLASHERB : TIMER := (PRE := 500, ACC := 202, EN := 1, TT := 1);   // Lamp Flasher Reset
   I : DINT[200];   // Integer Data
   IntegerTransferIndex : DINT;   // Index Register for Transfer of Integer Data to HMI
   IntegerTransferIndex2 : DINT;
   Oneshots : BOOL[128] := ([0] := 1, [13] := 1);
   RecordFault : BOOL;
   RecordPieceSaw1 : BOOL;   // Record Piece Count For Shift Total
   RecordPieceSaw2 : BOOL;   // Record Piece Count For Shift Total
   Rollcase1RunHourTimer : TIMER := (PRE := 360000);   // Rollcase 1 Run Hourmeter 1/10th Hour Timer
   Rollcase2RunHourTimer : TIMER := (PRE := 360000);   // Rollcase 2 Run Hourmeter 1/10th Hour Timer
   Saw1FailureDelay : TIMER := (PRE := 1000);
   Saw1RunHourTimer : TIMER := (PRE := 360000);   // Saw 1 Run Hourmeter 1/10th Hour Timer
   Saw2FailureDelay : TIMER := (PRE := 1000);
   Saw2RunHourTimer : TIMER := (PRE := 360000);   // Saw 2 Run Hourmeter 1/10th Hour Timer
   SplashScreen : TIMER := (PRE := 10000);
   T : TIMER[100] := ([2].PRE := 300, [3].PRE := 300, [6].ACC := 34, [6].EN := 1, [6].DN := 1, [7].PRE := 1000, [7].ACC := 1026, [7].EN := 1, [7].DN := 1, [10].PRE := 500, [11].PRE := 500, [12].ACC := 11, [12].EN := 1, [12].TT := 1, [13].PRE := 100, [19].PRE := 500, [20].PRE := 100, [21].PRE := 40, [22].PRE := 3000, [30].PRE := 1000, [31].PRE := 3000, [32].PRE := 1000, [33].PRE := 3000, [35].PRE := 2500, [39].PRE := 200, [40].PRE := 150, [41].ACC := 34, [41].EN := 1, [41].DN := 1, [44].PRE := 3000, [69].PRE := 500, [70].PRE := 100, [71].PRE := 40, [72].PRE := 3000, [89].PRE := 200, [90].PRE := 150, [91].PRE := 4000, [91].ACC := 4019, [91].EN := 1, [91].DN := 1, [94].PRE := 3000);   // Timers
        [6]   // Rollcase 1 VSD Power On Delay
        [13]   // Delay for Measurement
        [35]   // ChainEjector Watchodog Timer
        [19]   // Rollcase 1 Stop Delay
        [69]   // Rollcase 2 Stop Delay
        [39]   // PE Infeed Saw 1 Debounce
        [44]   // Saw 1 Feed OK Status Delay Timer
        [20]   // Rollcase 1 Stopping Delay
        [10]   // Reset Failure Pulse Timer
        [11]   // Reset Failure Pulse Timer
        [12]   // Cancel Reset Buffer Pulse Timer
        [89]   // PE Infeed Saw 2 Debounce
        [2]   // Pulse to Saw Computer Buffer Data to Saw 1
        [3]   // Pulse to Saw Computer Buffer Data to Saw 2
        [41]   // Saw 1 is Clear
        [91]   // Saw 2 is Clear
        [98]   // Saw 2 Infeed Blockage Delay
        [90]   // Saw 2 PE Debounce Timber Entering Saw
        [94]   // Saw 2 Feed OK Status Delay Timer
        [40]   // Saw 1 PE Debounce Timber Entering Saw
        [70]   // Rollcase Stopping Delay
        [71]   // Saw 2 Timber Ready Delay
        [21]   // Saw 1 Timber Ready Delay
        [72]   // Cross Feed 2 Watch Dog Timer
        [22]   // Cross Feed 1 Watchdog Timer
   TimerTransferIndex : DINT := 100;   // Index Register For Copying Timer Presets to HMI
   WasteBelt1RunHourTimer : TIMER := (PRE := 360000);   // Waste Belt 1 Run Hourmeter 1/10th Hour Timer
   WasteBelt2RunHourTimer : TIMER := (PRE := 360000);   // Waste Belt 2 Run Hourmeter 1/10th Hour Timer
END_VAR

ROUTINE BitTransferFromHMI   (* ladder *)
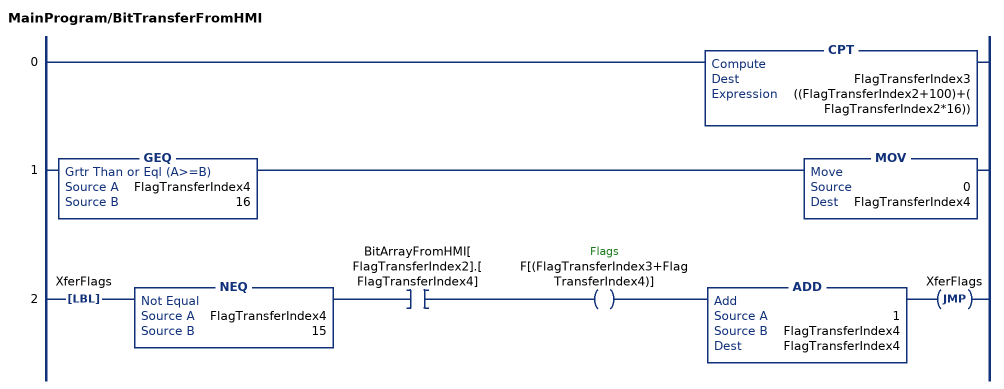
   0: CPT(FlagTransferIndex3,((FlagTransferIndex2+100)+(FlagTransferIndex2*16)));
   1: GEQ(FlagTransferIndex4,16)MOV(0,FlagTransferIndex4);
   2: LBL(XferFlags)NEQ(FlagTransferIndex4,15)XIC(BitArrayFromHMI[FlagTransferIndex2].[FlagTransferIndex4])OTE(F[(FlagTransferIndex3+FlagTransferIndex4)])ADD(1,FlagTransferIndex4,FlagTransferIndex4)JMP(XferFlags);
END_ROUTINE

ROUTINE BitTransferToHMI   (* ladder *)
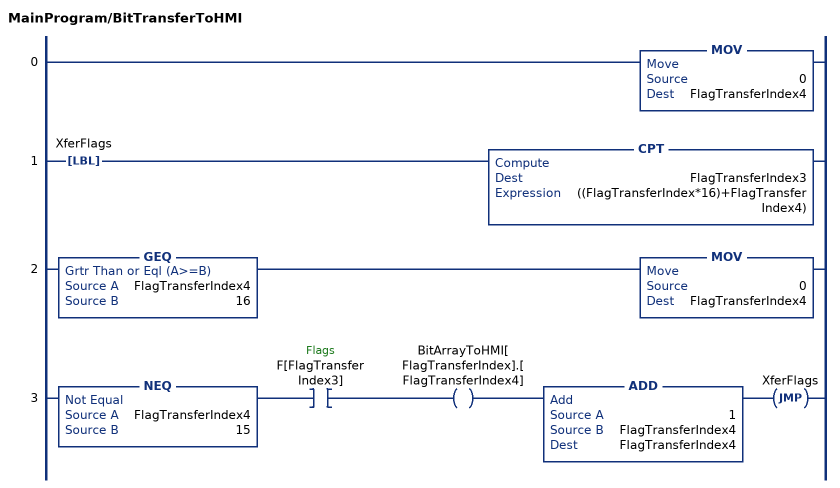
   0: MOV(0,FlagTransferIndex4);
   1: LBL(XferFlags)CPT(FlagTransferIndex3,((FlagTransferIndex*16)+FlagTransferIndex4));
   2: GEQ(FlagTransferIndex4,16)MOV(0,FlagTransferIndex4);
   3: NEQ(FlagTransferIndex4,15)XIC(F[FlagTransferIndex3])OTE(BitArrayToHMI[FlagTransferIndex].[FlagTransferIndex4])ADD(1,FlagTransferIndex4,FlagTransferIndex4)JMP(XferFlags);
END_ROUTINE

ROUTINE BufferControl   (* ladder *)
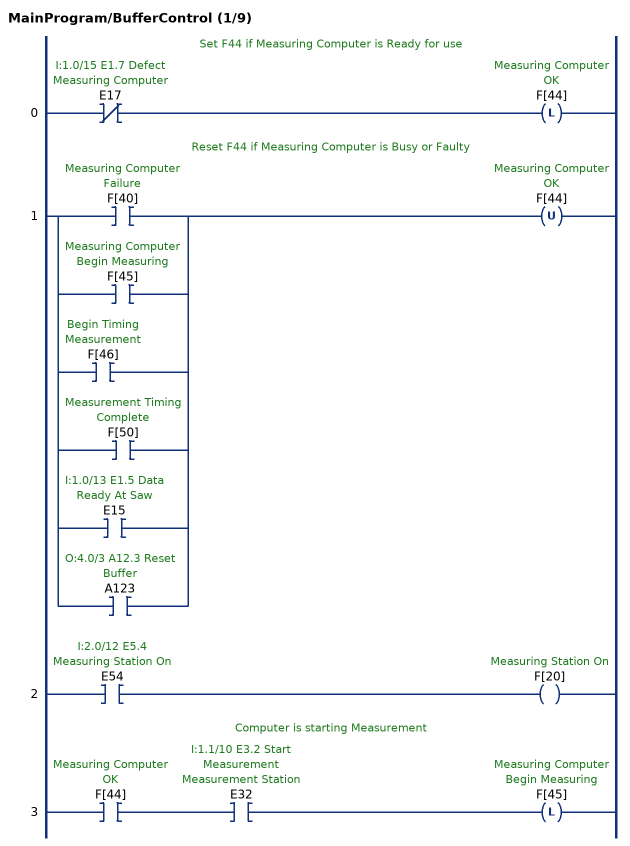
   // Set F44 if Measuring Computer is Ready for use
   0: XIO(E17)OTL(F[44]);
   // Reset F44 if Measuring Computer is Busy or Faulty
   1: [XIC(F[40]) ,XIC(F[45]) ,XIC(F[46]) ,XIC(F[50]) ,XIC(E15) ,XIC(A123) ]OTU(F[44]);
   2: XIC(E54)OTE(F[20]);
   // Computer is starting Measurement
   3: XIC(F[44])XIC(E32)OTL(F[45]);
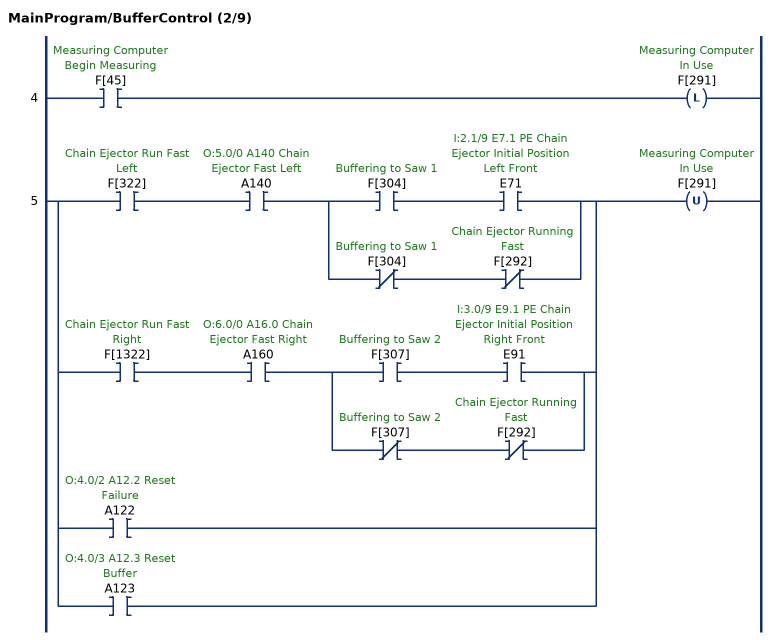
   4: XIC(F[45])OTL(F[291]);
   5: [XIC(F[322]) XIC(A140) [XIC(F[304]) XIC(E71) ,XIO(F[304]) XIO(F[292]) ] ,XIC(F[1322]) XIC(A160) [XIC(F[307]) XIC(E91) ,XIO(F[307]) XIO(F[292]) ] ,XIC(A122) ,XIC(A123) ]OTU(F[291]);
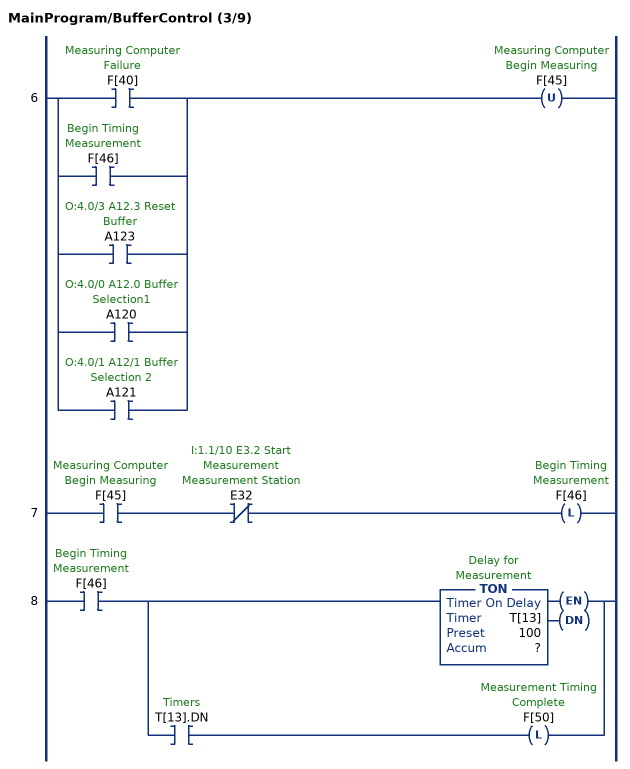
   6: [XIC(F[40]) ,XIC(F[46]) ,XIC(A123) ,XIC(A120) ,XIC(A121) ]OTU(F[45]);
   7: XIC(F[45])XIO(E32)OTL(F[46]);
   8: XIC(F[46])[TON(T[13],?,?) ,XIC(T[13].DN) OTL(F[50]) ];
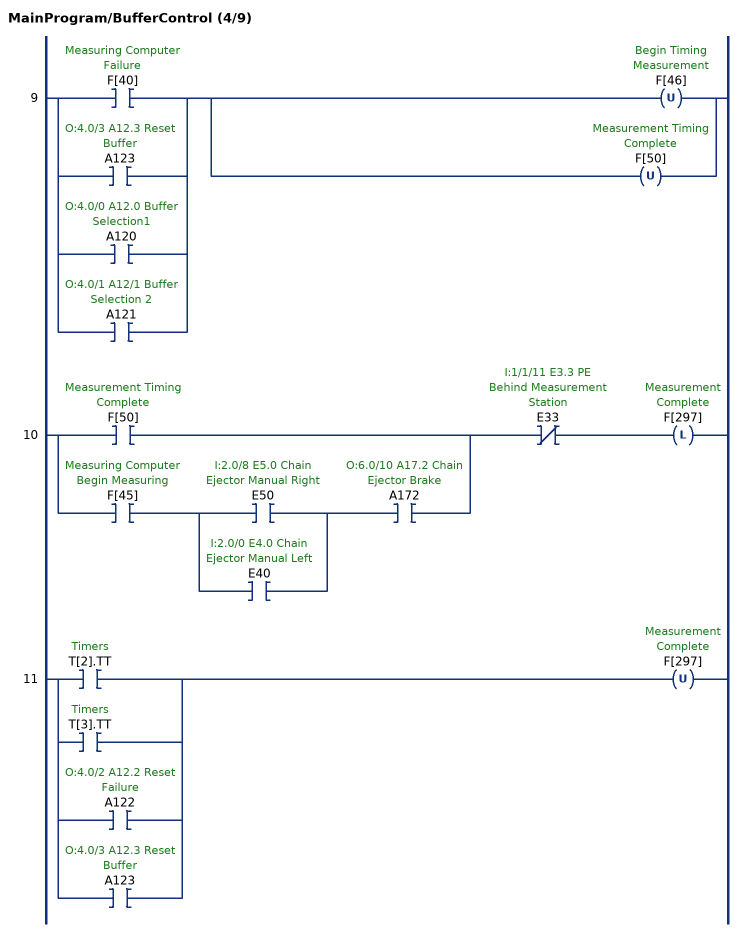
   9: [XIC(F[40]) ,XIC(A123) ,XIC(A120) ,XIC(A121) ][OTU(F[46]) ,OTU(F[50]) ];
   10: [XIC(F[50]) ,XIC(F[45]) [XIC(E50) ,XIC(E40) ] XIC(A172) ]XIO(E33)OTL(F[297]);
   11: [XIC(T[2].TT) ,XIC(T[3].TT) ,XIC(A122) ,XIC(A123) ]OTU(F[297]);
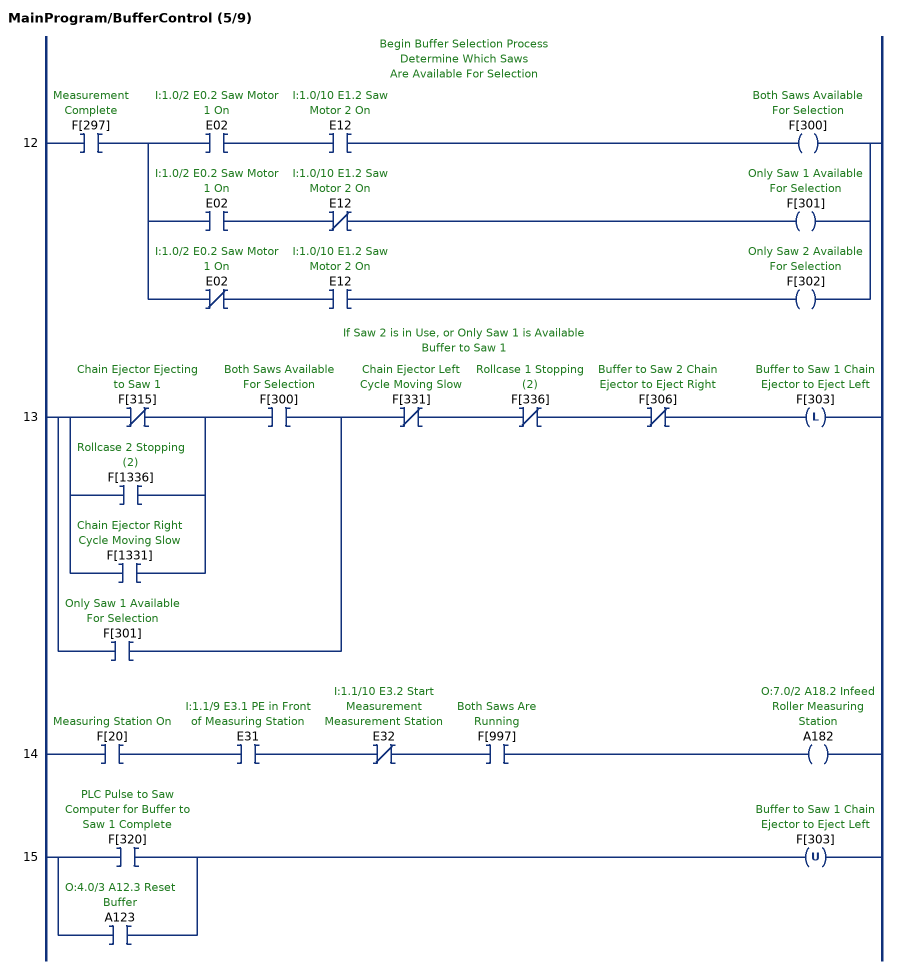
   // Begin Buffer Selection Process
   // Determine Which Saws
   // Are Available For Selection
   12: XIC(F[297])[XIC(E02) XIC(E12) OTE(F[300]) ,XIC(E02) XIO(E12) OTE(F[301]) ,XIO(E02) XIC(E12) OTE(F[302]) ];
   // If Saw 2 is in Use, or Only Saw 1 is Available
   // Buffer to Saw 1
   13: [[XIO(F[315]) ,XIC(F[1336]) ,XIC(F[1331]) ] XIC(F[300]) ,XIC(F[301]) ]XIO(F[331])XIO(F[336])XIO(F[306])OTL(F[303]);
   14: XIC(F[20])XIC(E31)XIO(E32)XIC(F[997])OTE(A182);
   15: [XIC(F[320]) ,XIC(A123) ]OTU(F[303]);
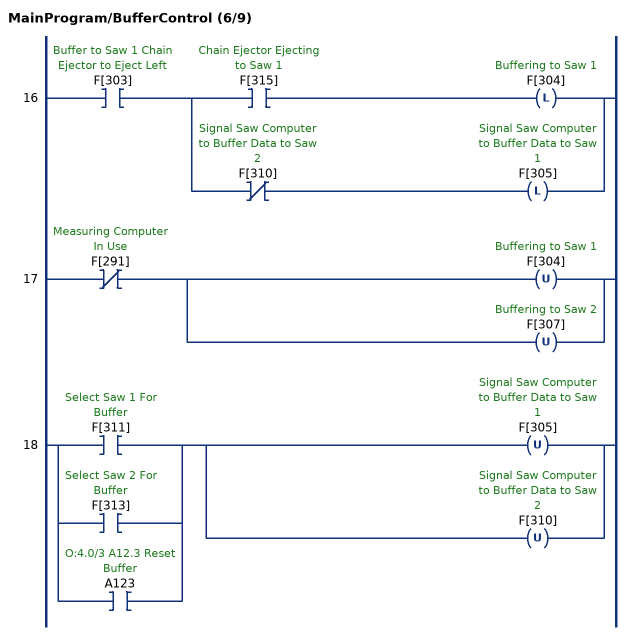
   16: XIC(F[303])[XIC(F[315]) OTL(F[304]) ,XIO(F[310]) OTL(F[305]) ];
   17: XIO(F[291])[OTU(F[304]) ,OTU(F[307]) ];
   18: [XIC(F[311]) ,XIC(F[313]) ,XIC(A123) ][OTU(F[305]) ,OTU(F[310]) ];
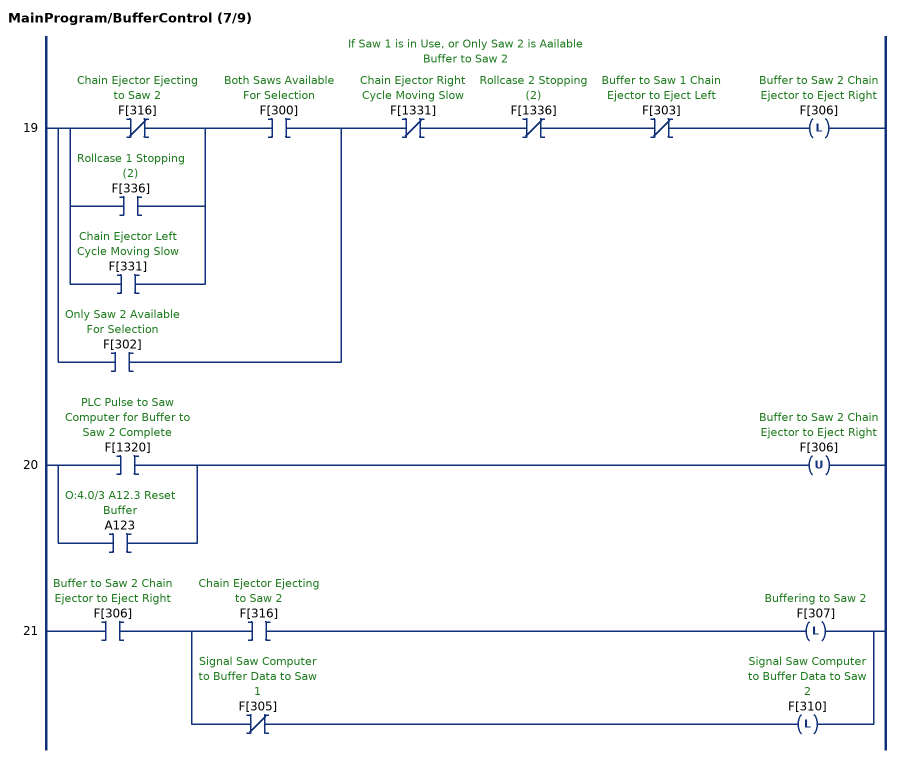
   // If Saw 1 is in Use, or Only Saw 2 is Aailable
   // Buffer to Saw 2
   19: [[XIO(F[316]) ,XIC(F[336]) ,XIC(F[331]) ] XIC(F[300]) ,XIC(F[302]) ]XIO(F[1331])XIO(F[1336])XIO(F[303])OTL(F[306]);
   20: [XIC(F[1320]) ,XIC(A123) ]OTU(F[306]);
   21: XIC(F[306])[XIC(F[316]) OTL(F[307]) ,XIO(F[305]) OTL(F[310]) ];
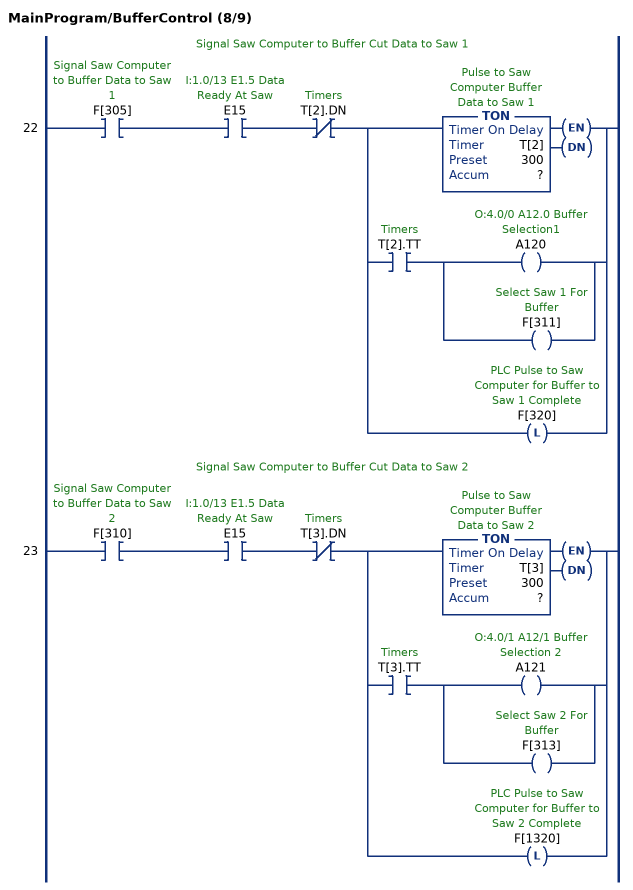
   // Signal Saw Computer to Buffer Cut Data to Saw 1
   22: XIC(F[305])XIC(E15)XIO(T[2].DN)[TON(T[2],?,?) ,XIC(T[2].TT) [OTE(A120) ,OTE(F[311]) ] ,OTL(F[320]) ];
   // Signal Saw Computer to Buffer Cut Data to Saw 2
   23: XIC(F[310])XIC(E15)XIO(T[3].DN)[TON(T[3],?,?) ,XIC(T[3].TT) [OTE(A121) ,OTE(F[313]) ] ,OTL(F[1320]) ];
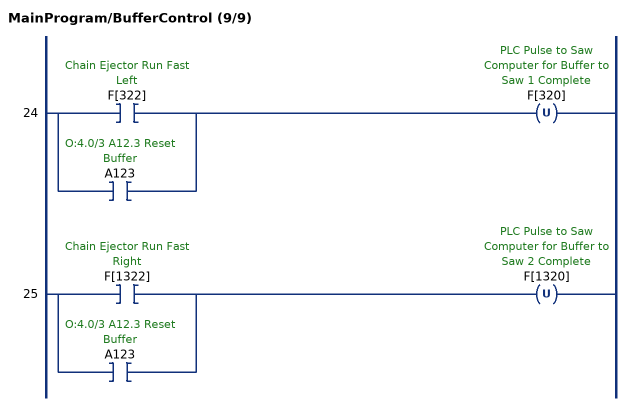
   24: [XIC(F[322]) ,XIC(A123) ]OTU(F[320]);
   25: [XIC(F[1322]) ,XIC(A123) ]OTU(F[1320]);
END_ROUTINE

ROUTINE ChainEjectors   (* ladder *)
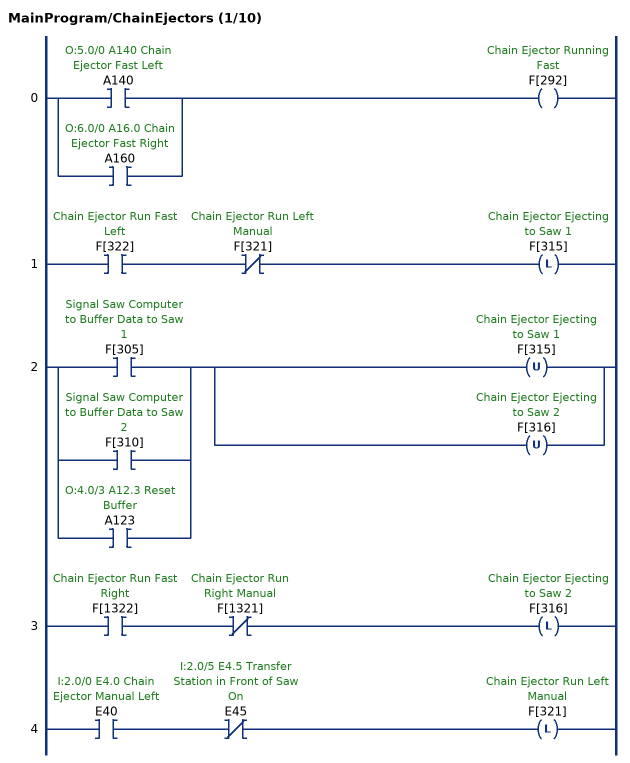
   0: [XIC(A140) ,XIC(A160) ]OTE(F[292]);
   1: XIC(F[322])XIO(F[321])OTL(F[315]);
   2: [XIC(F[305]) ,XIC(F[310]) ,XIC(A123) ][OTU(F[315]) ,OTU(F[316]) ];
   3: XIC(F[1322])XIO(F[1321])OTL(F[316]);
   4: XIC(E40)XIO(E45)OTL(F[321]);
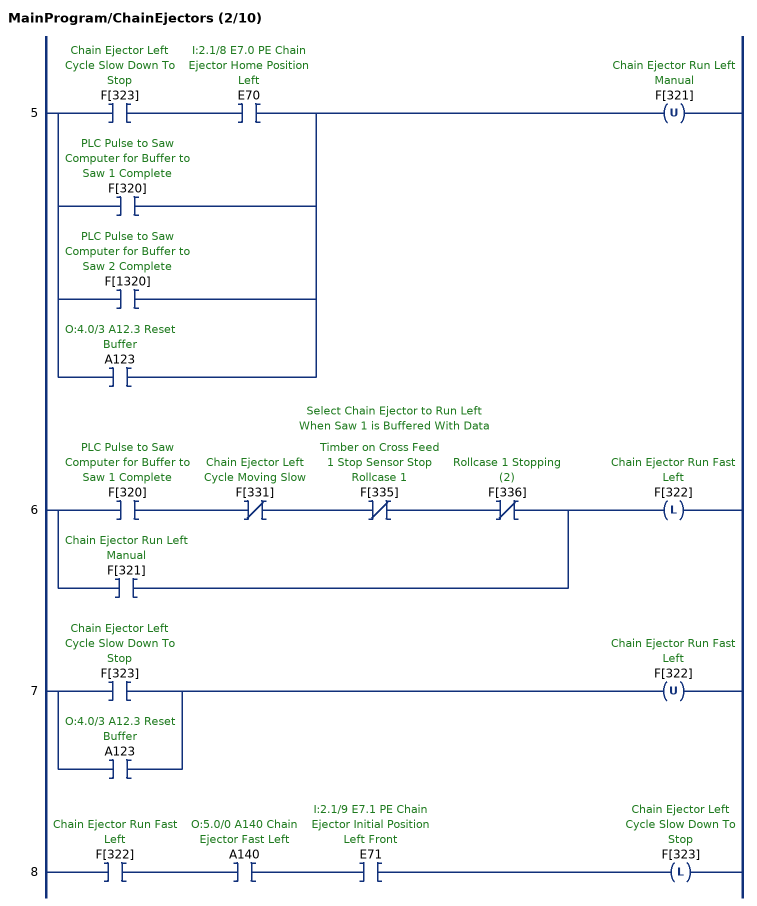
   5: [XIC(F[323]) XIC(E70) ,XIC(F[320]) ,XIC(F[1320]) ,XIC(A123) ]OTU(F[321]);
   // Select Chain Ejector to Run Left
   // When Saw 1 is Buffered With Data
   6: [XIC(F[320]) XIO(F[331]) XIO(F[335]) XIO(F[336]) ,XIC(F[321]) ]OTL(F[322]);
   7: [XIC(F[323]) ,XIC(A123) ]OTU(F[322]);
   8: XIC(F[322])XIC(A140)XIC(E71)OTL(F[323]);
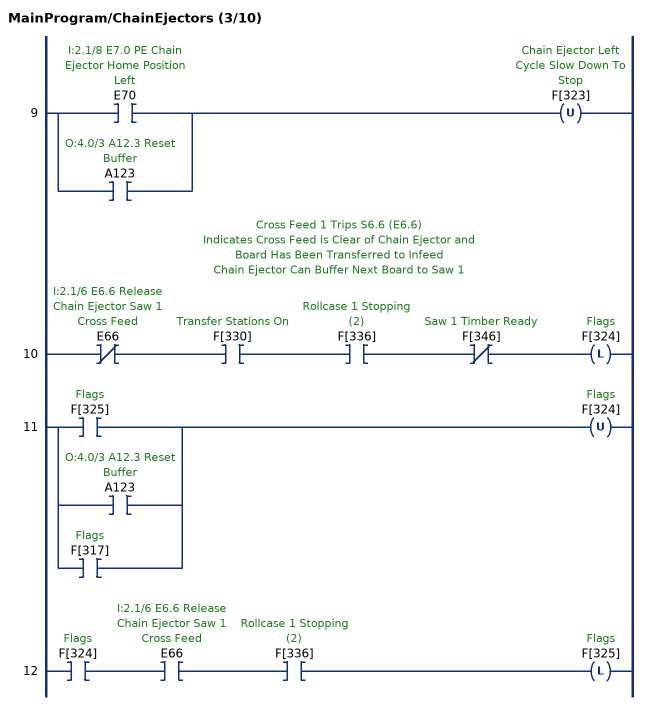
   9: [XIC(E70) ,XIC(A123) ]OTU(F[323]);
   // Cross Feed 1 Trips S6.6 (E6.6)
   // Indicates Cross Feed is Clear of Chain Ejector and
   // Board Has Been Transferred to Infeed
   // Chain Ejector Can Buffer Next Board to Saw 1
   10: XIO(E66)XIC(F[330])XIC(F[336])XIO(F[346])OTL(F[324]);
   11: [XIC(F[325]) ,XIC(A123) ,XIC(F[317]) ]OTU(F[324]);
   12: XIC(F[324])XIC(E66)XIC(F[336])OTL(F[325]);
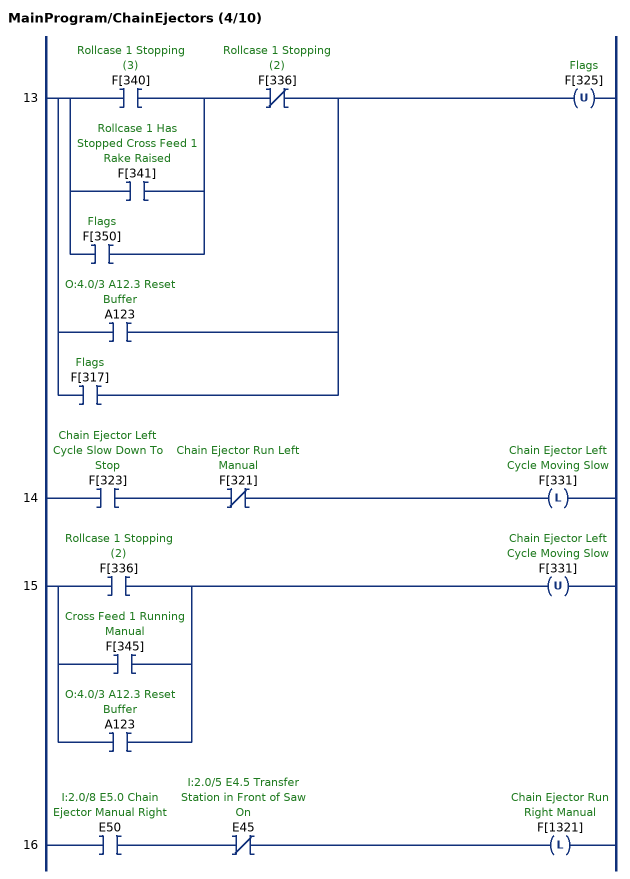
   13: [[XIC(F[340]) ,XIC(F[341]) ,XIC(F[350]) ] XIO(F[336]) ,XIC(A123) ,XIC(F[317]) ]OTU(F[325]);
   14: XIC(F[323])XIO(F[321])OTL(F[331]);
   15: [XIC(F[336]) ,XIC(F[345]) ,XIC(A123) ]OTU(F[331]);
   16: XIC(E50)XIO(E45)OTL(F[1321]);
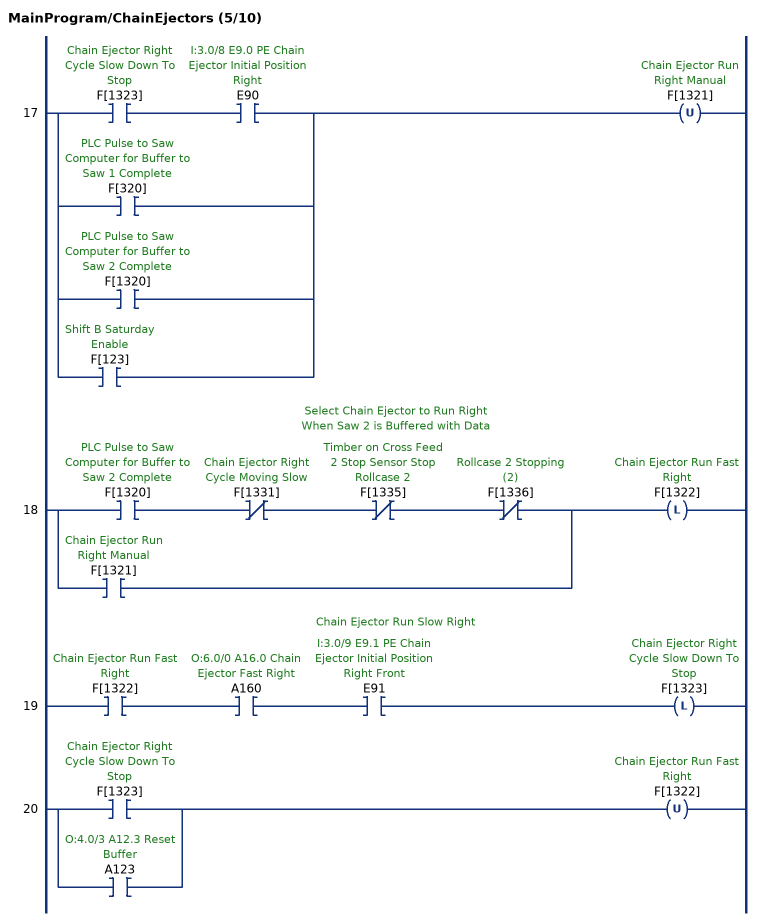
   17: [XIC(F[1323]) XIC(E90) ,XIC(F[320]) ,XIC(F[1320]) ,XIC(F[123]) ]OTU(F[1321]);
   // Select Chain Ejector to Run Right
   // When Saw 2 is Buffered with Data
   18: [XIC(F[1320]) XIO(F[1331]) XIO(F[1335]) XIO(F[1336]) ,XIC(F[1321]) ]OTL(F[1322]);
   // Chain Ejector Run Slow Right
   19: XIC(F[1322])XIC(A160)XIC(E91)OTL(F[1323]);
   20: [XIC(F[1323]) ,XIC(A123) ]OTU(F[1322]);
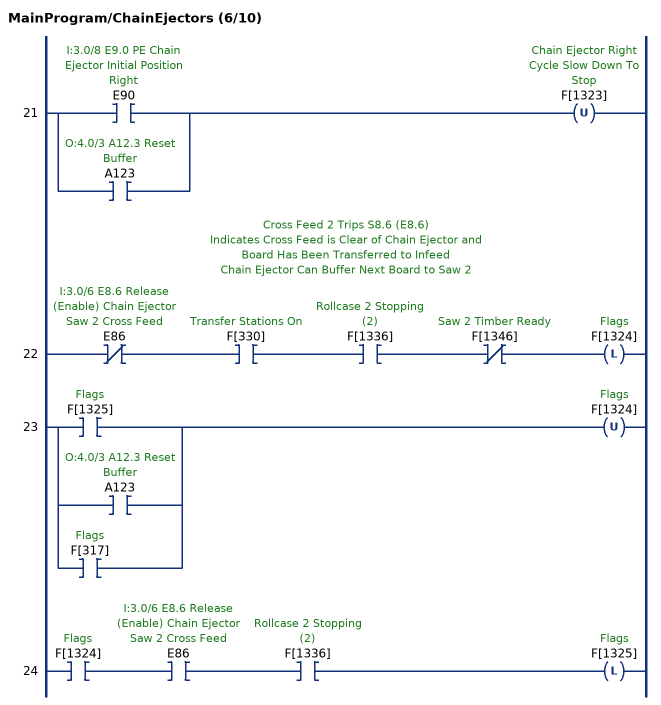
   21: [XIC(E90) ,XIC(A123) ]OTU(F[1323]);
   // Cross Feed 2 Trips S8.6 (E8.6)
   // Indicates Cross Feed is Clear of Chain Ejector and
   // Board Has Been Transferred to Infeed
   // Chain Ejector Can Buffer Next Board to Saw 2
   22: XIO(E86)XIC(F[330])XIC(F[1336])XIO(F[1346])OTL(F[1324]);
   23: [XIC(F[1325]) ,XIC(A123) ,XIC(F[317]) ]OTU(F[1324]);
   24: XIC(F[1324])XIC(E86)XIC(F[1336])OTL(F[1325]);
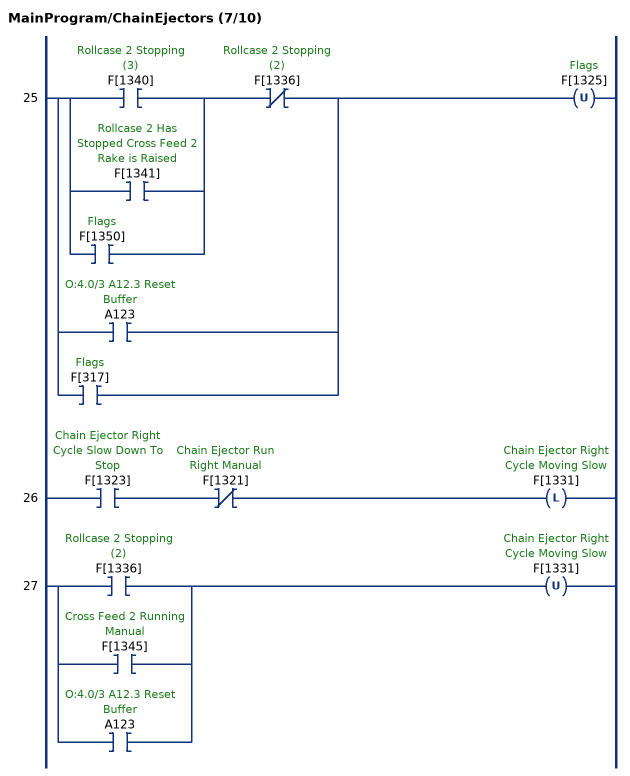
   25: [[XIC(F[1340]) ,XIC(F[1341]) ,XIC(F[1350]) ] XIO(F[1336]) ,XIC(A123) ,XIC(F[317]) ]OTU(F[1325]);
   26: XIC(F[1323])XIO(F[1321])OTL(F[1331]);
   27: [XIC(F[1336]) ,XIC(F[1345]) ,XIC(A123) ]OTU(F[1331]);
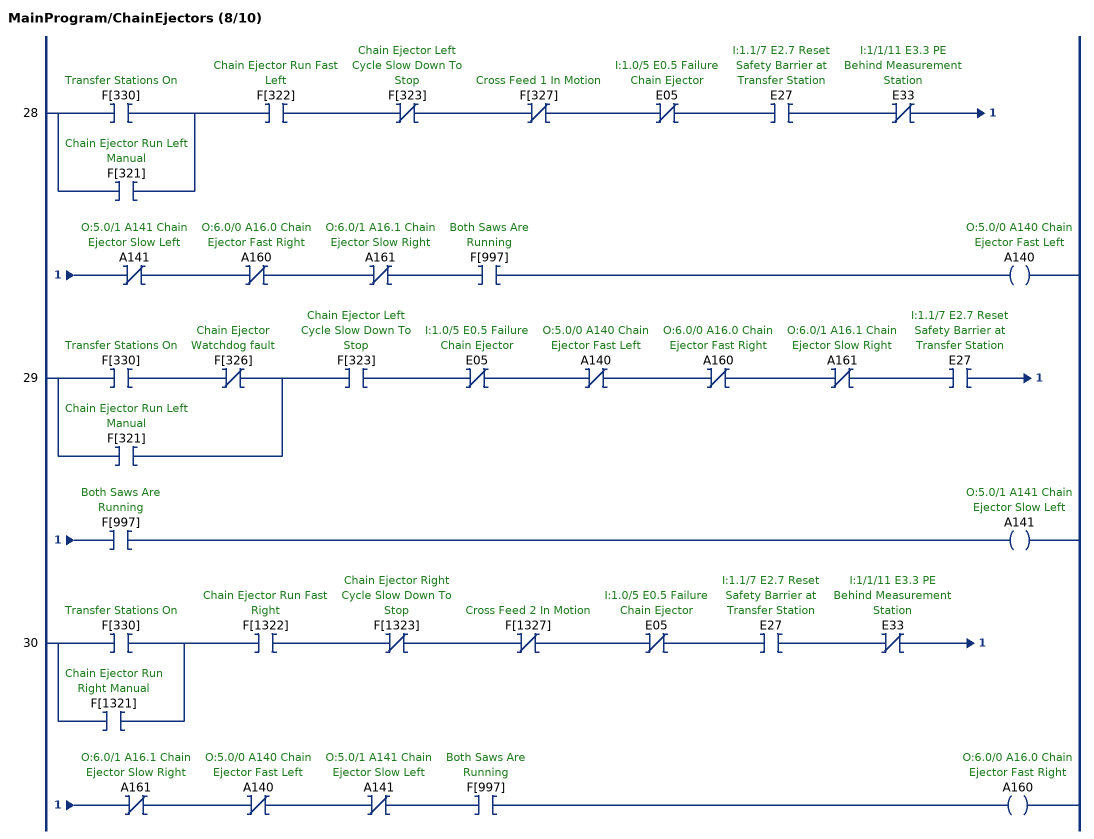
   28: [XIC(F[330]) ,XIC(F[321]) ]XIC(F[322])XIO(F[323])XIO(F[327])XIO(E05)XIC(E27)XIO(E33)XIO(A141)XIO(A160)XIO(A161)XIC(F[997])OTE(A140);
   29: [XIC(F[330]) XIO(F[326]) ,XIC(F[321]) ]XIC(F[323])XIO(E05)XIO(A140)XIO(A160)XIO(A161)XIC(E27)XIC(F[997])OTE(A141);
   30: [XIC(F[330]) ,XIC(F[1321]) ]XIC(F[1322])XIO(F[1323])XIO(F[1327])XIO(E05)XIC(E27)XIO(E33)XIO(A161)XIO(A140)XIO(A141)XIC(F[997])OTE(A160);
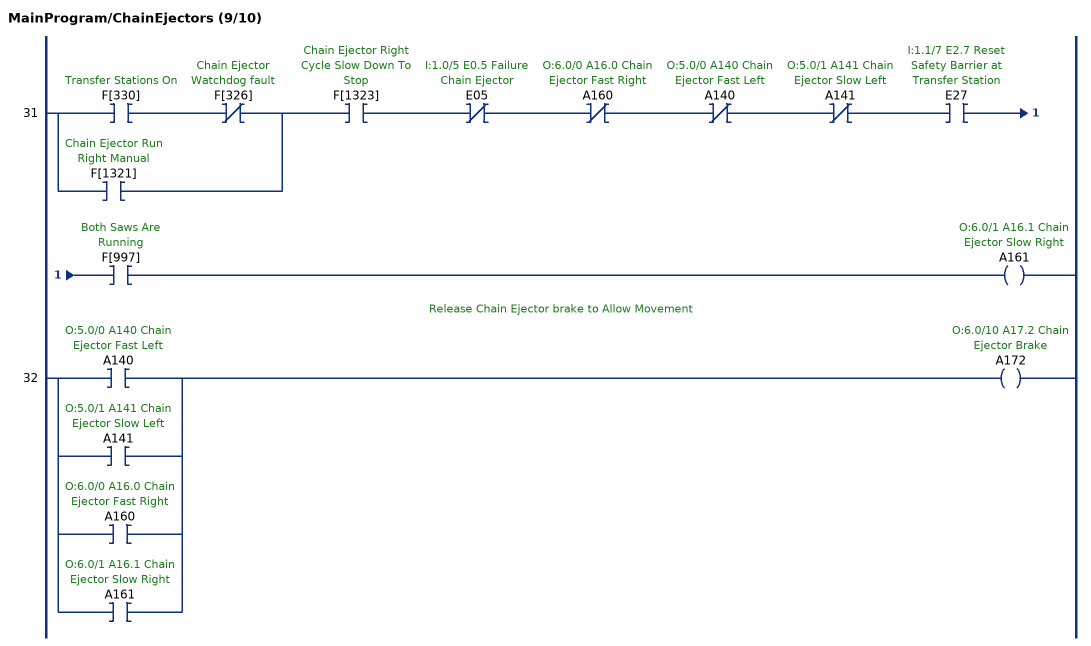
   31: [XIC(F[330]) XIO(F[326]) ,XIC(F[1321]) ]XIC(F[1323])XIO(E05)XIO(A160)XIO(A140)XIO(A141)XIC(E27)XIC(F[997])OTE(A161);
   // Release Chain Ejector brake to Allow Movement
   32: [XIC(A140) ,XIC(A141) ,XIC(A160) ,XIC(A161) ]OTE(A172);
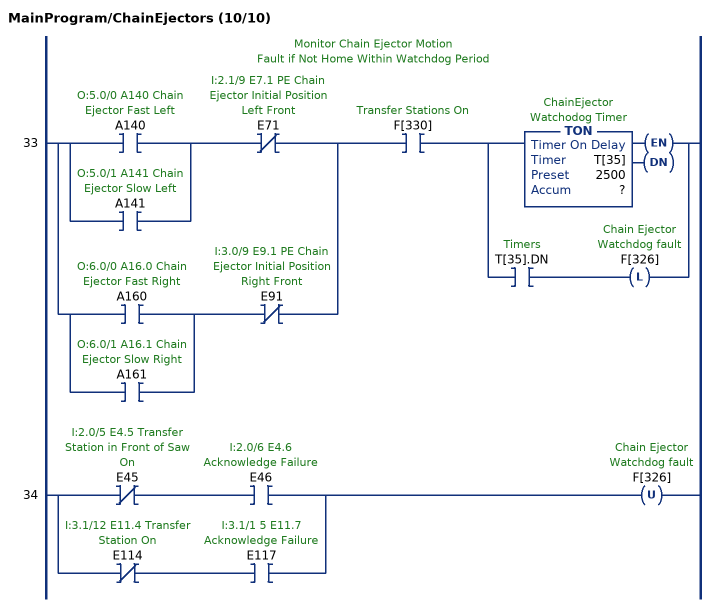
   // Monitor Chain Ejector Motion
   // Fault if Not Home Within Watchdog Period
   33: [[XIC(A140) ,XIC(A141) ] XIO(E71) ,[XIC(A160) ,XIC(A161) ] XIO(E91) ]XIC(F[330])[TON(T[35],?,?) ,XIC(T[35].DN) OTL(F[326]) ];
   34: [XIO(E45) XIC(E46) ,XIO(E114) XIC(E117) ]OTU(F[326]);
END_ROUTINE
